FUNCTION_BLOCK NormallyOpenSensor IMPLEMENTS I_Sensor
VAR
	input AT%I* : BOOL;
END_VAR

PROPERTY PUBLIC isActive : BOOL
GET
isActive	:=	input;
END_GET
END_PROPERTY

PROPERTY PUBLIC isInactive : BOOL
GET
isInactive	:=	NOT input;
END_GET
END_PROPERTY

END_FUNCTION_BLOCK

(* stored: Version 1.1.0.1, ProductVersion 3.1.4024.12
   POU NormallyOpenSensor: Id {0ade046d-2a77-424c-b21d-b10321ec10fd}, SpecialFunc None
   Property isActive: Id {e91573b4-fddd-4149-88fd-9a30f4f81c83}
   Get Get: Id {b95b4c13-4ff1-46fb-9897-29f1defb6736}
   Property isInactive: Id {01207b55-b113-49ca-b33d-2e3a704e73be}
   Get Get: Id {47fc47e5-c446-4959-9b16-7521cc9feec4} *)
